Staubli VAL3: onRun.pgx

public program onRun(string& x_sItem[])
  local bool l_bDone
  local string l_sItem
begin
  //
  // show the string
  //
  do
    if taskStatus("PULSE")==-1
      taskCreate "PULSE",20,execute(x_sItem,bExecute)
      watch(bExecute,0.5)
      l_bDone=true
    elseIf taskStatus("PULSE2")==-1
      taskCreate "PULSE2",20,execute(x_sItem,bExecute[1])
      watch(bExecute[1],0.5)
      l_bDone=true
    elseIf taskStatus("PULSE3")==-1
      taskCreate "PULSE3",20,execute(x_sItem,bExecute[2])
      watch(bExecute[2],0.5)
      l_bDone=true
    endIf
    delay(0)
  until l_bDone==true
end
